FUNCTION_BLOCK FB_MotionLogger_TestDouble IMPLEMENTS I_MotionLogger
VAR
END_VAR

END_FUNCTION_BLOCK

(* stored: Version 1.1.0.1
   POU FB_MotionLogger_TestDouble: Id {8442344f-b7dd-4d6a-a684-1fd8fe76a797}, SpecialFunc None *)
